INTERFACE I_Mode

METHOD Auto
VAR_INPUT
	bAuto : BOOL;
END_VAR
END_METHOD

METHOD Manual
VAR_INPUT
	bManual : BOOL;
END_VAR
END_METHOD

METHOD Off
VAR_INPUT
	bEnabled : BOOL;
END_VAR
END_METHOD

END_INTERFACE

(* stored: Version 1.1.0.1, ProductVersion 3.1.4024.10
   Itf I_Mode: Id {251fceed-e838-489a-8a0d-24a86c22225d}
   Method Auto: Id {0fd1d885-6f37-46c1-a51e-05fd717f4a37}
   Method Manual: Id {24373131-a1ad-403d-b2b4-b32be369fc78}
   Method Off: Id {44924819-9d1f-4d07-b949-7eb3ff82412a} *)
